(* LS Electric XG5000 project: OR AND *)
(* PLC LSPLC *)
(* module base 0 slot 0: 입력 모듈:XGI-D22A/B (DC 24V 입력, 16점 (전류소스 싱크공용/ 전류소스 입력)) *)
(* module base 0 slot 1: 입력 모듈:XGI-D22A/B (DC 24V 입력, 16점 (전류소스 싱크공용/ 전류소스 입력)) *)
(* module base 0 slot 2: 출력 모듈:XGQ-RY2A/B (릴레이 출력, 16점 (2A용, Varistor 없음/Varistor 부착)) *)
(* module base 0 slot 3: 출력 모듈:XGQ-RY2A/B (릴레이 출력, 16점 (2A용, Varistor 없음/Varistor 부착)) *)

PROGRAM NewProgram (* task: 스캔 프로그램 *)
VAR
    D1 : TIME;
    P0 : BOOL;
    T1 : TON;
    T2 : TON;
    이순신 : BOOL;
END_VAR

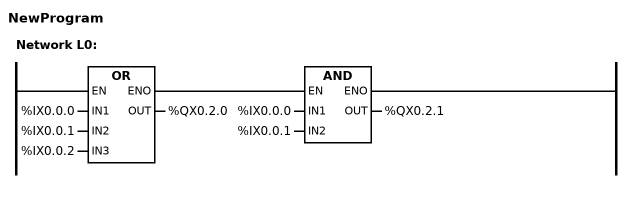
(* Rung L0 *)
%QX0.2.0 := %IX0.0.0 OR %IX0.0.1 OR %IX0.0.2;
%QX0.2.1 := %IX0.0.0 AND %IX0.0.1;
END_PROGRAM